FUNCTION_BLOCK Collection_Mockup EXTENDS Collection
VAR
END_VAR

METHOD GetItemByIndex : I_Base
VAR_INPUT
	Index : UDINT;
END_VAR

VAR
	pItem : POINTER TO I_Base;
END_VAR
pItem		   := Collection.pBuffer + (Index * SIZEOF(PVOID));
GetItemByIndex := pItem^;
END_METHOD

END_FUNCTION_BLOCK

(* stored: Version 1.1.0.1, ProductVersion 3.1.4026.18
   POU Collection_Mockup: Id {0df1fef0-f1a2-4c84-94bd-311358ab686f}, SpecialFunc None
   Method GetItemByIndex: Id {ee8270c2-cf91-4b72-8356-5206c8e1dc89} *)
